// TIA Portal project "Buong_chan_khong" (V14)

(* hardware
DEVICE "HMI_1"  KTP700 Basic PN
   slot 0: "KTP700 Basic PN"  KTP700 Basic PN  6AV2 123-2GB03-0AX0  14.0.1.0
   slot 1: "HMI_RT_1"  KTP700 Basic PN  6AV2 123-2GB03-0AX0  14.0.1.0
   slot 5: "HMI_1.IE_CP_1"  PROFINET Interface  14.0.1.0
      slot 1: "PROFINET Interface_1"  PROFINET Interface
         slot 1: "Port_1"  Port
DEVICE "S7-1200 station_1"  S7-1200 Station
   slot 0: "Rack_0"  S7-1200 Rack  Rack  V1.0
   slot 1: "PLC_1"  CPU 1214C DC/DC/DC  6ES7 214-1AG40-0XB0  V4.2
*)

// ===== PLC "PLC_1"  CPU 1214C DC/DC/DC =====

VAR_GLOBAL   // PLC tag table "Default tag table"
   "Congtac" AT %M0.0 : Bool;
   "buong" AT %Q0.0 : Bool;
   "System_Byte" AT %MB1 : Byte;
   "FirstScan" AT %M1.0 : Bool;
   "DiagStatusUpdate" AT %M1.1 : Bool;
   "AlwaysTRUE" AT %M1.2 : Bool;
   "AlwaysFALSE" AT %M1.3 : Bool;
   "Clock_Byte" AT %MB0 : Byte;
   "Clock_10Hz" AT %M0.0 : Bool;
   "Clock_5Hz" AT %M0.1 : Bool;
   "Clock_2.5Hz" AT %M0.2 : Bool;
   "Clock_2Hz" AT %M0.3 : Bool;
   "Clock_1.25Hz" AT %M0.4 : Bool;
   "Clock_1Hz" AT %M0.5 : Bool;
   "Clock_0.625Hz" AT %M0.6 : Bool;
   "Clock_0.5Hz" AT %M0.7 : Bool;
   "System_Byte(1)" AT %MB1 : Byte;
   "System_Byte(2)" AT %MB1 : Byte;
   "Tag_1" AT %IW64 : Int;
   "Tag_2" AT %MD10 : Real;
   "Tag_3" AT %MD14 : Real;
   "CD1" AT %Q0.1 : Bool;
   "Tag_4" AT %IW32 : Int;
   "Tag_5" AT %MD11 : Real;
   "Tag_6" AT %MD15 : Real;
   "CD2" AT %Q0.2 : Bool;
   "CTbuong" AT %I0.0 : Bool;
   "CD3" AT %Q0.3 : Bool;
   "CT" AT %M2.0 : Bool;
   "Tag_7" AT %IW66 : Int;
   "Start" AT %M2.1 : Bool;
   "Flag" AT %M2.2 : Bool;
   "Tag_8" AT %Q0.4 : Bool;
END_VAR

// folder: System blocks/Program resources

DATA_BLOCK "IEC_Timer_0_DB"   // DB1
{ S7_Optimized_Access := 'TRUE' }
AUTHOR : Simatic
FAMILY : IEC
NAME : IEC_TMR
VERSION : 1.0
// stored: InstanceOfName IEC_TIMER
"IEC_TIMER"
BEGIN
END_DATA_BLOCK

DATA_BLOCK "IEC_Timer_0_DB_1"   // DB2
{ S7_Optimized_Access := 'TRUE' }
AUTHOR : Simatic
FAMILY : IEC
NAME : IEC_TMR
VERSION : 1.0
// stored: InstanceOfName IEC_TIMER
"IEC_TIMER"
BEGIN
END_DATA_BLOCK

// folder: (top level)

ORGANIZATION_BLOCK "Main"   // OB1, LAD, ProgramCycle
TITLE = "Main Program Sweep (Cycle)"
{ S7_Optimized_Access := 'TRUE' }
VERSION : 0.1
   VAR_INPUT
      Initial_Call : Bool;   // Initial call of this OB
      Remanence : Bool;   // =True, if remanent data are available
   END_VAR
   VAR_TEMP   // added for the SCL form of the ladder/FBD networks
      _w1 : Bool;
   END_VAR
BEGIN

REGION Network 1
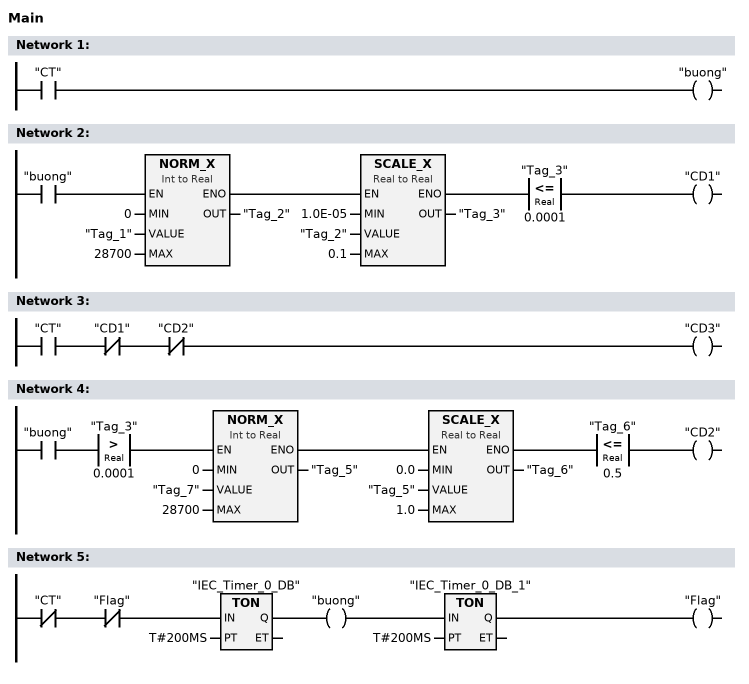
   RUNG wire#powerrail
      Contact( "CT" )
      Coil( "buong" )
   END_RUNG
   // the same network as SCL:
   "buong" := "CT";
END_REGION

REGION Network 2
   RUNG wire#powerrail
      Contact( "buong" )
      { S7_Templates := "[SrcType := Int, DestType := Real]" } Normalize(min := 0, value := "Tag_1", max := 28700, out => "Tag_2")
      { S7_Templates := "[SrcType := Real, DestType := Real]" } Scale(min := 1.0E-05, value := "Tag_2", max := 0.1, out => "Tag_3")
      { S7_Templates := "SrcType := Real" } LE_Contact(in1 := "Tag_3", in2 := 0.0001)
      Coil( "CD1" )
   END_RUNG
   // the same network as SCL:
   IF "buong" THEN
       "Tag_2" := NORM_X(MIN := 0, VALUE := "Tag_1", MAX := 28700);
       "Tag_3" := SCALE_X(MIN := 1.0E-05, VALUE := "Tag_2", MAX := 0.1);
   END_IF;
   "CD1" := "buong" AND ("Tag_3" <= 0.0001);
END_REGION

REGION Network 3
   RUNG wire#powerrail
      Contact( "CT" )
      I_Contact( "CD1" )
      I_Contact( "CD2" )
      Coil( "CD3" )
   END_RUNG
   // the same network as SCL:
   "CD3" := "CT" AND NOT "CD1" AND NOT "CD2";
END_REGION

REGION Network 4
   RUNG wire#powerrail
      Contact( "buong" )
      { S7_Templates := "SrcType := Real" } GT_Contact(in1 := "Tag_3", in2 := 0.0001)
      { S7_Templates := "[SrcType := Int, DestType := Real]" } Normalize(min := 0, value := "Tag_7", max := 28700, out => "Tag_5")
      { S7_Templates := "[SrcType := Real, DestType := Real]" } Scale(min := 0.0, value := "Tag_5", max := 1.0, out => "Tag_6")
      { S7_Templates := "SrcType := Real" } LE_Contact(in1 := "Tag_6", in2 := 0.5)
      Coil( "CD2" )
   END_RUNG
   // the same network as SCL:
   #_w1 := "buong" AND ("Tag_3" > 0.0001);
   IF #_w1 THEN
       "Tag_5" := NORM_X(MIN := 0, VALUE := "Tag_7", MAX := 28700);
       "Tag_6" := SCALE_X(MIN := 0.0, VALUE := "Tag_5", MAX := 1.0);
   END_IF;
   "CD2" := #_w1 AND ("Tag_6" <= 0.5);
END_REGION

REGION Network 5
   "IEC_Timer_0_DB".TON(IN := NOT "CT" AND NOT "Flag", PT := T#200MS);
   "buong" := "IEC_Timer_0_DB".Q;
   "IEC_Timer_0_DB_1".TON(IN := "IEC_Timer_0_DB".Q, PT := T#200MS);
   "Flag" := "IEC_Timer_0_DB_1".Q;
END_REGION
END_ORGANIZATION_BLOCK

(* ===== HMI "HMI_RT_1" =====
system functions are stored by id; their names below are inferred from use
connection "HMI_Connection_1": ETHERNET, SMART_S7_1200_OMS

HMI tags "Default tag table"
   "Tag_ScreenNumber" : UInt, internal
   "Tag_6" : Real = PLC Tag_6 AT %MD15, 1 s
   "Tag_2" : Real = PLC Tag_2 AT %MD10, 1 s
   "CT" : Bool = PLC CT AT %M2.0, 1 s
   "buong" : Bool = PLC buong AT %Q0.0, 1 s
   "Tag_3" : Real = PLC Tag_3 AT %MD14, 1 s
   "CD1" : Bool = PLC CD1 AT %Q0.1, 1 s
   "CD2" : Bool = PLC CD2 AT %Q0.2, 1 s
   "CD3" : Bool = PLC CD3 AT %Q0.3, 1 s
   "Tag_8" : Bool = PLC Tag_8 AT %Q0.4, 1 s

Template "Template_1" 800x480
   Button "Exit" at 714,429 size 71x50; TextOff 'Exit'; PictureOff "ExitRuntime_KTP700_Basic_PN_TR"; PictureOn "ExitRuntime_KTP700_Basic_PN_TR"
      on Release: StopRuntime(0)
   Button "Template_Button" at 614,429 size 71x50; TextOff 'Text'
   Button "Template_Button_1" at 514,429 size 71x50; TextOff 'Text'
   Button "Template_Button_2" at 414,429 size 71x50; TextOff 'Text'
   Button "Template_Button_3" at 314,429 size 71x50; TextOff 'Text'
   Button "Template_Button_4" at 214,429 size 71x50; TextOff 'Text'
   Button "Template_Button_5" at 114,429 size 71x50; TextOff 'Text'
   Button "Start screen" at 14,429 size 71x50; TextOff 'Start screen'; PictureOff "NavigateHome_KTP700_Basic_PN_TR"; PictureOn "NavigateHome_KTP700_Basic_PN_TR"
      on Release: ActivateScreen("Root screen", 0)
   SymbolicIOField "Symbolic_IO_Field_Screen" at 93,9 size 600x33; TextOff '0'; TextOn '1'; TextList "TextList_ScreenNames"
      ProcessValue <- "Tag_ScreenNumber"
      on Change: ActivateScreenByNumber("Tag_ScreenNumber", 0)
   DateTimeField "HmiScreenItemData" at 695,25 size 105x25
   DateTimeField "HmiScreenItemData_1" at 695,0 size 105x25
   GraphicView "Logo" at 0,0 size 91x51; Picture "Logo of HMI_1"

screen "Root screen" 800x480, template "Template_1"
   on GenerateScreen: SetTag("Tag_ScreenNumber", 1)
   Button "Button_1" at 67,200 size 192x32; TextOff 'Cong_doan_1'
      on Click: ActivateScreen("Cong_doan_1", 0)
   Button "Button_2" at 67,265 size 192x32; TextOff 'Cong_doan_2'
      on Click: ActivateScreen("Cong_doan_2", 0)
   Button "Button_3" at 67,330 size 192x32; TextOff 'Cong_doan_3'
      on Click: ActivateScreen("Cong_doan_3", 0)
   Circle "Circle_1" at 195,84 size 84x84
      Appearance <- "buong"
   Switch "Switch_1" at 75,117 size 80x32; CaptionText 'Switch'; TextOff 'OFF'; TextOn 'ON'
      on SwitchOn: SetBit("CT")
      on SwitchOff: ResetBit("CT")
   TextField "Text field_1" at 215,116 size 37x23; Text 'Đèn'
   Circle "Circle_2" at 322,199 size 30x30
      Appearance <- "CD1"
   Circle "Circle_3" at 322,265 size 30x30
      Appearance <- "CD2"
   Circle "Circle_4" at 322,331 size 30x30
      Appearance <- "CD3"
   Circle "Circle_5" at 549,142 size 45x45
      Appearance <- "Tag_8"

screen "Cong_doan_3" 800x480
   Button "Button_1" at 533,44 size 192x32; TextOff 'Root screen'
      on Click: ActivateScreen("Root screen", 0)
   Circle "Circle_4" at 245,91 size 30x30
      Appearance <- "CD3"

screen "Cong_doan_2" 800x480
   Button "Button_1" at 554,55 size 192x32; TextOff 'Root screen'
      on Click: ActivateScreen("Root screen", 0)
   Bar "Bar_1" at 112,51 size 145x337; MinimumValue 0; MaximumValue 1
      ProcessValue <- "Tag_6"
   IOField "I/O field_1" at 299,169 size 96x32; FormatPattern s99.999
      ProcessValue <- "Tag_6"
   Circle "Circle_3" at 523,190 size 56x56
      Appearance <- "CD2"

screen "Cong_doan_1" 800x480
   Bar "Bar_1" at 160,20 size 102x226; MinimumValue 1e-05; MaximumValue 0.1
      ProcessValue <- "Tag_3"
   IOField "I/O field_1" at 303,131 size 96x32; FormatPattern s9.999
      ProcessValue <- "Tag_3"
   Button "Button_1" at 546,45 size 192x32; TextOff 'Root screen'
      on Click: ActivateScreen("Root screen", 0)
   Circle "Circle_1" at 311,218 size 71x71
      Appearance <- "CD1"
*)